// SIMATIC S7-200 project (STEP 7-Micro/WIN), CPU 221 REL 01.10

SYMBOL_TABLE USR1
Always_On        SM0.0    // This bit is always on.
Write_Date       I0.0     // Operate the switch at input I0.0 to write preset date to the real time clock.
Change_Code      I0.1     // Select BCD format (I0.1 = 1) or binary format (I0.1 = 0).
Second_Display   QB0      // The seconds in the real-time clock are displayed at output Q0.0
END_SYMBOL_TABLE

ORGANIZATION_BLOCK MAIN:OB1
TITLE=
// 怎样读和写S7-200的实时时钟
// ***概述***
// 这个程序示例涉及到关于实时时钟的两种特殊指令：读和写日期及时钟时间。
// 为了进行这些操作，需要有如下结构的8字节缓冲区：
// 字节0： 年（00-99）  字节4： 分（00-59）
// 字节1： 月（1-12）   字节5： 秒（00-59）
// 字节2： 日（1-31）   字节6： 未分配
// 字节3： 时（00-24）  字节7： 星期（1-7=Su-Sa）
// 为了读或写方便，这些数据用BCD码存储。当操作开关I0.0为1时，就将预定日期和
// 时间写入实时时钟。为了显示当前的秒值，将其值拷贝到输出字节QB0.当I0.1=1时，
// 则用BCD码显示；当I0.1=0时，则用二进制码显示。
// ***程序和注释***
// 通过按输入开关I0.0，可调用子程序0。这个子程序按照要求的时间和日期，预先将
// 其值置入VB100到VB107这8个字节，然后用TODW指令，将此设置传送给实时时钟
// 每个周期都读出实时时钟的值，这些数据以BCD码形式（4位代表0-9的数字）存储在
// VB400到VB407这8个字节中。如果输入I0.1为1，这些值就被直接拷贝到输出字节QB0,
// 以供显示。
// 如果输入开关I0.1为0，将数据从VW404拷贝到VW204,再将包含分钟值的VW204清零。
// 这一步是必须的，因为把秒值从BCD码的形式转换成二进制码的形式，只能按字来转换。
// 现时的二进制码的秒值被传输到输出字节QB0,以供显示。
// 
BEGIN
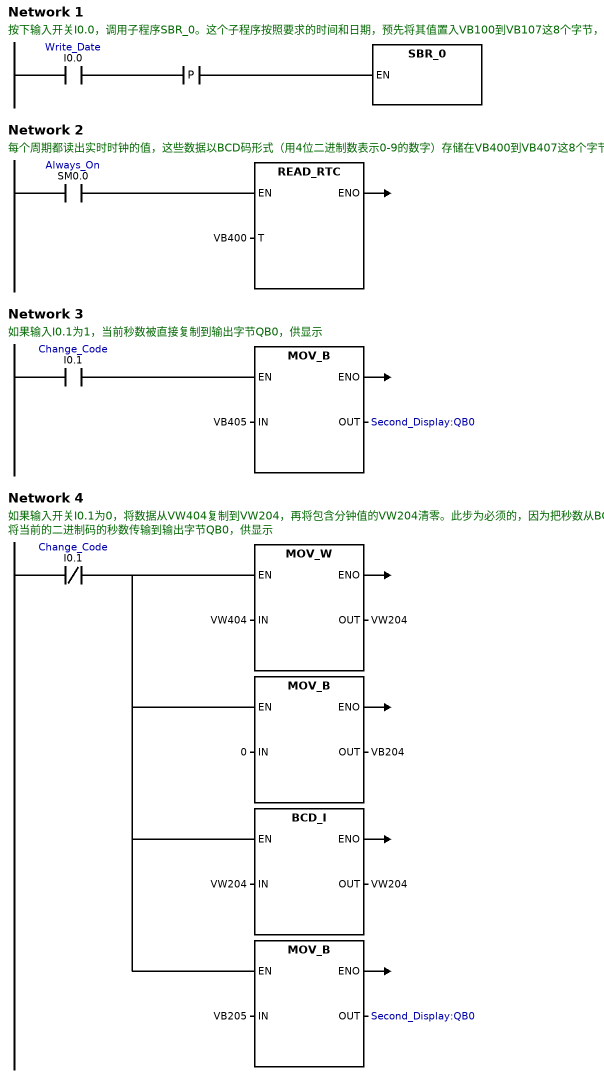
Network 1
// 按下输入开关I0.0，调用子程序SBR_0。这个子程序按照要求的时间和日期，预先将其值置入VB100到VB107这8个字节，将此设置传送给实时时钟
// 写实时时钟的开关，若按I0.0开头
// 上升沿，则
// 调用子程序0，写实时时钟
LD     Write_Date:I0.0
EU
CALL   SBR_0:SBR0
Network 2
// 每个周期都读出实时时钟的值，这些数据以BCD码形式（用4位二进制数表示0-9的数字）存储在VB400到VB407这8个字节中
// 设置栈顶
// 读出实时时钟数据并填入8字节
//缓冲区（VB400至VB407）
LD     Always_On:SM0.0
TODR   VB400
Network 3
// 如果输入I0.1为1，当前秒数被直接复制到输出字节QB0，供显示
// 以BCD码的形式显示秒的开关，若I0.1=1,则
// 将当前秒值拷贝到输出字节QB0
LD     Change_Code:I0.1
MOVB   VB405, Second_Display:QB0
Network 4
// 如果输入开关I0.1为0，将数据从VW404复制到VW204，再将包含分钟值的VW204清零。此步为必须的，因为把秒数从BCD码的形式转换成二进制码的形式，只能按字转换
// 将当前的二进制码的秒数传输到输出字节QB0，供显示
//以二进制码的形式显示秒的开关，若I0.1=0,则
// 将字VW404拷贝到字VW204
// 清除高字节VB204(分)
// BCD码转换为二进制码（秒）
// 当前秒值拷贝到输出字节QB0
LDN    Change_Code:I0.1
MOVW   VW404, VW204
MOVB   0, VB204
BCDI   VW204
MOVB   VB205, Second_Display:QB0
Network 5 // 主程序结束
// MEND				
// 
Network 6 // ***子程序0***
END_ORGANIZATION_BLOCK

SUBROUTINE_BLOCK SBR_0:SBR0
TITLE=
BEGIN
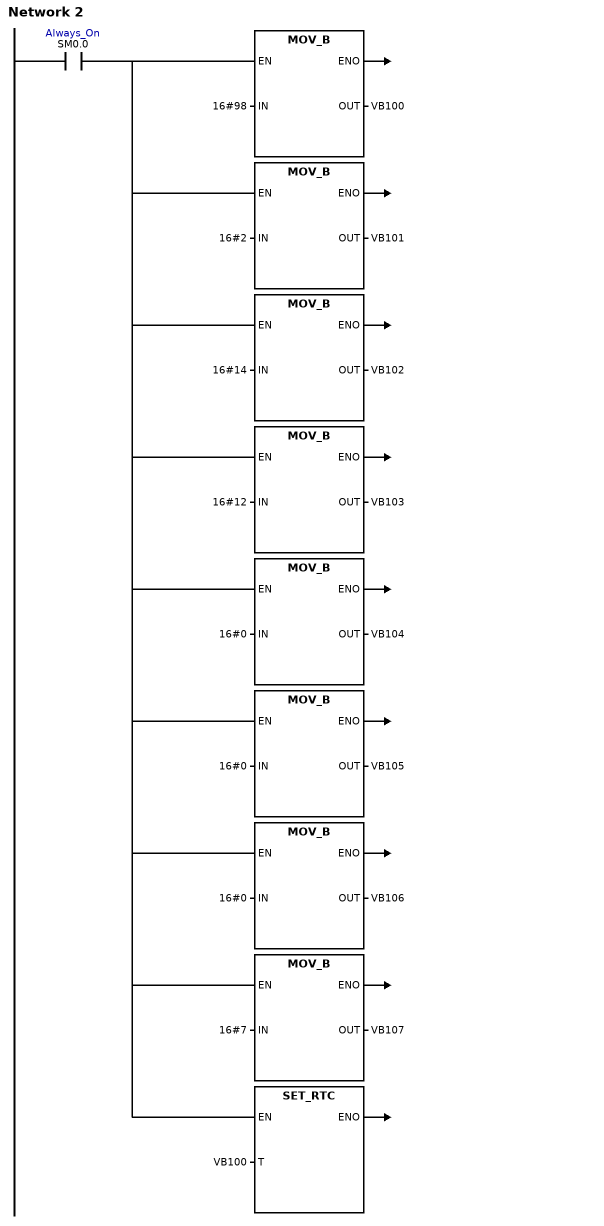
Network 2
// 年：98
// 月：2月
// 日：14
// 时：12
// 分： 00.
// 秒：00.
// 未分配
// 星期：Saturday.
// 写实时时钟
LD     Always_On:SM0.0
MOVB   16#98, VB100
MOVB   16#2, VB101
MOVB   16#14, VB102
MOVB   16#12, VB103
MOVB   16#0, VB104
MOVB   16#0, VB105
MOVB   16#0, VB106
MOVB   16#7, VB107
TODW   VB100
Network 3 // 子程序0结束
// RET					
// 
END_SUBROUTINE_BLOCK
